// manual Err_Ack 
GVL_Safety.ErrAck := (GVL_Main.key_switch_remote AND GVL_Main.reset_switch);

// manual Restart
GVL_Safety.Restart := (GVL_Main.key_switch_remote AND GVL_Main.start_switch);

ErrAckLog(	Trigger := GVL_Safety.ErrAck,
			OnMessage := 'Safety error was acknowledged.');
			
RestartLog(	Trigger := GVL_Safety.Restart,
			Level := ADSLOG_MSGTYPE_WARN,
			OnMessage := 'Safety was restarted.');

SafetyLog(	Trigger := Error,
			Level := ADSLOG_MSGTYPE_ERROR,
			OnMessage := 'Safety Error! Emergency stop enganged!',
			OffMessage := 'Safety is OK.',
			OffLevel := ADSLOG_MSGTYPE_HINT);
*)

(*
// wait n seconds after Start ...
start_delay(IN := TRUE);
// ... and send ErrAck for n milliseconds
ErrAck_Pulse(IN := (GVL_Safety.State = 2) AND start_delay.Q);

// Error Acknowledgment: Turn key_switch OFF and press STOP 
GVL_Safety.ErrAck := (GVL_Main.key_switch_remote AND GVL_Main.reset_switch)
					OR ErrAck_Pulse.Q
					OR remote_ErrAck;
// detect falling edge 
ErrAck_Trigger(CLK := GVL_Safety.ErrAck);
// send restart pulse on falling edge of ErrAck
restart_pulse(IN := ErrAck_Trigger.Q);

// RESTART Safety after pushing reset or power on delay
GVL_Safety.Restart := (GVL_Main.key_switch_remote AND GVL_Main.start_switch)
 					   OR remote_restart
                       OR restart_pulse.Q;
				
//Error := GVL_Safety.Error OR (GVL_Safety.State <> 1);

//Emergency_stop := NOT GVL_Safety.Stop;

ErrAckLog(	Trigger := GVL_Safety.ErrAck,
			OnMessage := 'Safety error was acknowledged.');
			
RestartLog(	Trigger := GVL_Safety.Restart,
			Level := ADSLOG_MSGTYPE_WARN,
			OnMessage := 'Safety was restarted.');

SafetyLog(	Trigger := Error,
			Level := ADSLOG_MSGTYPE_ERROR,
			OnMessage := 'Safety Error! Emergency stop enganged!',
			OffMessage := 'Safety is OK.',
			OffLevel := ADSLOG_MSGTYPE_HINT);
*)

END_PROGRAM

// ---- POUs/FunctionBlocks/FB_InfoGroup.TcPOU
FUNCTION_BLOCK FB_InfoGroup
VAR_INPUT
	stInfoData	:ST_InfoDataGroup;
END_VAR
VAR_OUTPUT
	sState		:STRING;
END_VAR
VAR
END_VAR

IF stInfoData.usiMapState= 1 THEN
	sState:='RUN';
ELSIF stInfoData.usiMapState= 2 THEN
	sState:='STOP';
ELSIF stInfoData.usiMapState= 3 THEN
	sState:='SAFE';
ELSIF stInfoData.usiMapState= 4 THEN
	sState:='ERROR';
ELSIF stInfoData.usiMapState= 5 THEN
	sState:='RESET';
ELSE
	sState:='Unknown';
END_IF

END_FUNCTION_BLOCK

// ---- POUs/FunctionBlocks/FB_InfoEStop.TcPOU
FUNCTION_BLOCK FB_InfoEStop
VAR_INPUT
	stInfoData		:ST_InfoDataFB;
END_VAR
VAR_OUTPUT
	sState			:STRING;
	sDiag			:STRING;
END_VAR

IF stInfoData.usiMapState= 0 THEN
	sState:='undefined';
ELSIF stInfoData.usiMapState= 1 THEN
	sState:='RUN';
ELSIF stInfoData.usiMapState= 2 THEN
	sState:='STOP';
ELSIF stInfoData.usiMapState= 3 THEN
	sState:='SAFE';
ELSIF stInfoData.usiMapState= 4 THEN
	sState:='ERROR';
ELSIF stInfoData.usiMapState= 5 THEN
	sState:='RESET';
ELSIF stInfoData.usiMapState= 6 THEN
	sState:='START';
ELSIF stInfoData.usiMapState= 8 THEN
	sState:='DELAYOUT';
ELSE
	sState:='Unknown';
END_IF

IF stInfoData.uiMapDiag = 0 THEN
	sDiag:='No error';
ELSIF stInfoData.uiMapDiag.0 THEN
	sDiag:='Discrepancy error input group 1';
ELSIF stInfoData.uiMapDiag.1 THEN
	sDiag:='Discrepancy error input group 2';
ELSIF stInfoData.uiMapDiag.2 THEN
	sDiag:='Discrepancy error input group 3';
ELSIF stInfoData.uiMapDiag.3 THEN
	sDiag:='Discrepancy error input group 4';
ELSIF stInfoData.uiMapDiag.4 THEN
	sDiag:='EDM Error EDM 1';
ELSIF stInfoData.uiMapDiag.5 THEN
	sDiag:='EDM Error EDM 2';
ELSE
	sDiag:='Unknown';
END_IF

END_FUNCTION_BLOCK

// ---- POUs/FunctionBlocks/FB_InfoConnection.TcPOU
FUNCTION_BLOCK FB_InfoConnection
VAR_INPUT
	stInfoData	:ST_InfoDataConnection;
END_VAR
VAR_OUTPUT
	sState		:STRING;
	sDiag		:STRING;
	bChannel1	:BOOL;
	bChannel2	:BOOL;
	bChannel3	:BOOL;
	bChannel4	:BOOL;
END_VAR

IF stInfoData.usiMapState = 100 THEN
	sState:='State Reset';
ELSIF stInfoData.usiMapState = 101 THEN
	sState:='State Session';
ELSIF stInfoData.usiMapState = 102 THEN
	sState:='State Connection';
ELSIF stInfoData.usiMapState = 103 THEN
	sState:='State Parameter';
ELSIF stInfoData.usiMapState = 104 THEN
	sState:='State Data';
ELSIF stInfoData.usiMapState = 105 THEN
	sState:='State Shutdown';
ELSE
	sState:='Error';
END_IF

IF stInfoData.usiMapDiag = 0 THEN
	sDiag:='No error';
ELSIF	stInfoData.usiMapDiag.0 = TRUE THEN
	sDiag:='Invalid Command';
ELSIF	stInfoData.usiMapDiag.1 = TRUE THEN
	sDiag:='Unknown Command';
ELSIF	(stInfoData.usiMapDiag.1 AND stInfoData.usiMapDiag.0)= TRUE THEN
	sDiag:='Invalid Connection ID';
ELSIF	 stInfoData.usiMapDiag.2= TRUE THEN
	sDiag:='Invalid CRC';
ELSIF	(stInfoData.usiMapDiag.0 AND stInfoData.usiMapDiag.2)= TRUE THEN
	sDiag:='Watchdog expired';
ELSIF	(stInfoData.usiMapDiag.1 AND stInfoData.usiMapDiag.2)= TRUE THEN
	sDiag:='Invalid FSoE address';
ELSIF	(stInfoData.usiMapDiag.0 AND stInfoData.usiMapDiag.1 AND stInfoData.usiMapDiag.2)= TRUE THEN
	sDiag:='Invalid data';
ELSIF	stInfoData.usiMapDiag.3= TRUE THEN
	sDiag:='Invalid Com.-Parameter length';
ELSIF	(stInfoData.usiMapDiag.0 AND stInfoData.usiMapDiag.3)= TRUE THEN
	sDiag:='Invalid Com.-Parameter ';
ELSIF	(stInfoData.usiMapDiag.1 AND stInfoData.usiMapDiag.3)= TRUE THEN
	sDiag:='Invalid User.-Parameter length';
ELSIF	(stInfoData.usiMapDiag.0 AND stInfoData.usiMapDiag.1 AND stInfoData.usiMapDiag.3)= TRUE THEN
	sDiag:='Invalid User.-Parameter ';
ELSIF	(stInfoData.usiMapDiag.2 AND stInfoData.usiMapDiag.3)= TRUE THEN
	sDiag:='FSoE Master Reset  ';
ELSIF	stInfoData.usiMapDiag.4= TRUE THEN
	sDiag:='Error by FSoE Slave detected';
ELSIF	stInfoData.usiMapDiag.5= TRUE THEN
	sDiag:='FSoE Slave reports Failsafe value active';
ELSIF	stInfoData.usiMapDiag.6= TRUE THEN
	sDiag:='StartUp';
ELSIF	stInfoData.usiMapDiag.7= TRUE THEN
	sDiag:='FSoE Master reports Failsafe value active';
ELSE
	sDiag:='Error';
END_IF

(*Signals*)
bChannel1 := stInfoData.bySignal.0;
bChannel2 := stInfoData.bySignal.1;
bChannel3 := stInfoData.bySignal.2;
bChannel4 := stInfoData.bySignal.3;

END_FUNCTION_BLOCK

// ---- GlobalTextList.TcGTLO
TEXTLIST GlobalTextList
  785 = 'Azimuth:'
  798 = 'Brake closed'
  396 = 'Brake open'
  272 = 'busy'
  41 = 'Close brake'
  815 = 'Derotator:'
  524 = 'Diag: %s'
  101 = 'EL1904'
  761 = 'EL2904'
  409 = 'Elevation:'
  894 = 'Enable'
  868 = 'ErrAck'
  879 = 'Error'
  225 = 'Estop: %s'
  548 = 'GoHome'
  867 = 'GoTo'
  33 = 'Oil cold'
  995 = 'Oil high'
  856 = 'Oil hot'
  768 = 'Oil low'
  481 = 'Oil pressure OK'
  498 = 'Oil warning'
  482 = 'Open brake'
  352 = 'Override Start Pump'
  744 = 'Override Start Sucction'
  606 = 'Override stop pump'
  273 = 'park'
  919 = 'Power'
  523 = 'Pump running'
  120 = 'ready'
  685 = 'Reset'
  789 = 'Restart'
  104 = 'Safety Diag%s'
  521 = 'Safety Diag: %s'
  672 = 'Safety State: %s'
  777 = 'slew'
  717 = 'sliding'
  809 = 'State: %s'
  328 = 'STO ErrAck:'
  540 = 'STO Reset:'
  488 = 'STO:'
  572 = 'Stop'
  155 = 'stopped'
  782 = 'Sucction running'
  704 = 'Succtionrunning'
  362 = 'track'
  364 = 'tracking'
END_TEXTLIST

// ---- VISUs/Safety.TcVIS
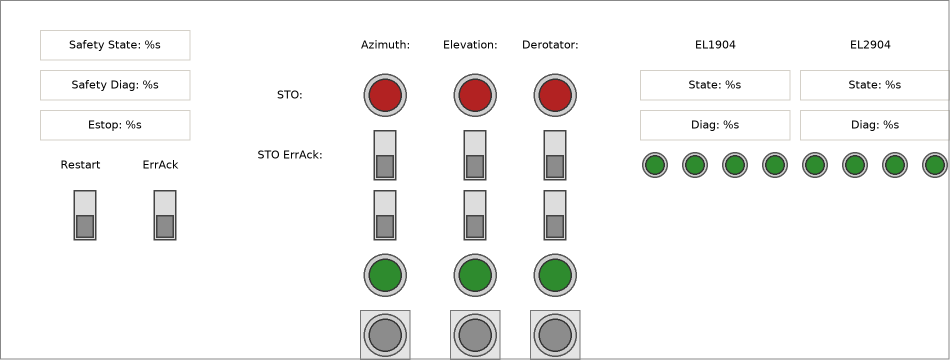
VISUALIZATION Safety  // 950x360
    Label (340,30 91x30), "Azimuth:"
    Lamp1 (360,70 50x50), variable: GVL_Telescope.Azimuth_sto, style: Lamp-Lamp1-Red
    Label (430,30 81x30), "Elevation:"
    Lamp1 (450,70 50x50), variable: GVL_Telescope.Elevation_sto, style: Lamp-Lamp1-Red
    Label (510,30 81x30), "Derotator:"
    Lamp1 (530,70 50x50), variable: GVL_Telescope.Derotator_sto, style: Lamp-Lamp1-Red
    Label (240,80 100x30), "STO:"
    Lamp1 (360,250 50x50), variable: AzimuthElevationControl.ready, style: Lamp-Lamp1-Green
    Lamp1 (450,250 50x50), variable: ElevationControl.Ready, style: Lamp-Lamp1-Green
    Lamp1 (530,250 50x50), style: Lamp-Lamp1-Green
    PushSwitch (360,310 50x50), variable: AzimuthElevationControl.Reset, behaviour: TAP, style: Switch-PushSwitch-Gray
    PushSwitch (450,310 50x50), variable: ElevationControl.reset, behaviour: TAP, style: Switch-PushSwitch-Gray
    PushSwitch (530,310 50x50), behaviour: TAP, style: Switch-PushSwitch-Gray
    DipSwitch (360,190 50x50), variable: AzimuthElevationControl.Enable, behaviour: TOGGLE, style: Switch-DipSwitch-Gray
    DipSwitch (450,190 50x50), variable: ElevationControl.enable, behaviour: TOGGLE, style: Switch-DipSwitch-Gray
    DipSwitch (530,190 50x50), variable: DerotatorControl.enable, behaviour: TOGGLE, style: Switch-DipSwitch-Gray
    DipSwitch (60,190 50x50), variable: GVL_Safety.Restart, behaviour: TOGGLE, style: Switch-DipSwitch-Gray
    DipSwitch (530,130 50x50), variable: GVL_Safety.Reset_STO_Derotator, behaviour: TOGGLE, style: Switch-DipSwitch-Gray
    DipSwitch (360,130 50x50), variable: GVL_Safety.Reset_STO_Azimuth, behaviour: TOGGLE, style: Switch-DipSwitch-Gray
    DipSwitch (450,130 50x50), variable: GVL_Safety.Reset_STO_Elevation, behaviour: TOGGLE, style: Switch-DipSwitch-Gray
    Label (240,140 100x30), "STO ErrAck:"
    Label (40,150 81x30), "Restart"
    DipSwitch (140,190 50x50), variable: GVL_Safety.ErrAck, behaviour: TOGGLE, style: Switch-DipSwitch-Gray
    Label (120,150 81x30), "ErrAck"
    Textfield (40,30 150x30), "Safety State: %s", text variable: SafetyHandling.fbInfoEStop1.sState, input disabled if: TRUE
    Textfield (40,110 150x30), "Estop: %s", text variable: SafetyHandling.fbInfoEStop1.sState, input disabled if: TRUE
    Textfield (40,70 150x30), "Safety Diag: %s", text variable: SafetyHandling.fbInfoEStop1.sDiag, input disabled if: TRUE
    Label (670,30 91x30), "EL1904"
    Label (830,30 81x30), "EL2904"
    Textfield (640,70 150x30), "State: %s", text variable: SafetyHandling.fbInfoSafetyIn.sState, input disabled if: TRUE
    Textfield (640,110 150x30), "Diag: %s", text variable: SafetyHandling.fbInfoSafetyIn.sDiag, input disabled if: TRUE
    Textfield (800,70 150x30), "State: %s", text variable: SafetyHandling.fbInfoSafetyOut.sState, input disabled if: TRUE
    Textfield (800,110 150x30), "Diag: %s", text variable: SafetyHandling.fbInfoSafetyOut.sDiag, input disabled if: TRUE
    Lamp1 (640,150 30x30), variable: SafetyHandling.bSafetyInCh1, style: Lamp-Lamp1-Green
    Lamp1 (680,150 30x30), variable: SafetyHandling.bSafetyInCh2, style: Lamp-Lamp1-Green
    Lamp1 (720,150 30x30), variable: SafetyHandling.bSafetyInCh3, style: Lamp-Lamp1-Green
    Lamp1 (760,150 30x30), variable: SafetyHandling.bSafetyInCh4, style: Lamp-Lamp1-Green
    Lamp1 (800,150 30x30), variable: SafetyHandling.bSafetyInCh1, style: Lamp-Lamp1-Green
    Lamp1 (840,150 30x30), variable: SafetyHandling.bSafetyInCh2, style: Lamp-Lamp1-Green
    Lamp1 (880,150 30x30), variable: SafetyHandling.bSafetyInCh3, style: Lamp-Lamp1-Green
    Lamp1 (920,150 30x30), variable: SafetyHandling.bSafetyInCh4, style: Lamp-Lamp1-Green
END_VISUALIZATION

// ---- VISUs/Visualization.TcVIS
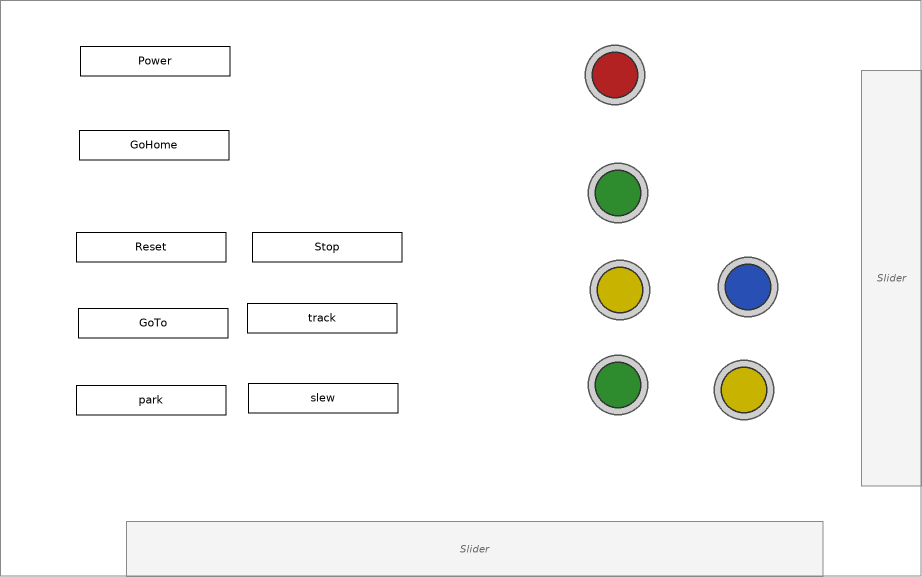
VISUALIZATION Visualization  // 922x577
    RoundedRectangle (80,46 150x30), "Power", colour toggle: TelescopeControl.power
        toggle TelescopeControl.power
    Rectangle (79,130 150x30), "GoHome", colour toggle: TelescopeControl.gohome
        toggle TelescopeControl.gohome
    Lamp1 (580,40 70x70), tooltip "Error", variable: TelescopeControl.error, style: Lamp-Lamp1-Red
    Lamp1 (583,158 70x70), tooltip "ready", variable: TelescopeControl.ready, style: Lamp-Lamp1-Green
    Rectangle (76,232 150x30), "Reset", colour toggle: TelescopeControl.reset
        toggle TelescopeControl.reset
    RoundedRectangle (78,308 150x30), "GoTo", colour toggle: TelescopeControl.goto
        toggle TelescopeControl.goto
    Lamp1 (585,255 70x70), tooltip "sliding", variable: TelescopeControl.sliding, style: Lamp-Lamp1-Yellow
    RoundedRectangle (76,385 150x30), "park", colour toggle: TelescopeControl.park
        toggle TelescopeControl.park
    Lamp1 (583,350 70x70), tooltip "stopped", variable: TelescopeControl.Safetypped, style: Lamp-Lamp1-Green
    Slider (126,521 697x56), variable: TelescopeControl.rightascension, scale 0..360
    Slider (861,70 61x416), variable: TelescopeControl.declination, scale -90..90
    Lamp1 (713,252 70x70), tooltip "tracking", variable: TelescopeControl.tracking, style: Lamp-Lamp1-Blue
    RoundedRectangle (247,303 150x30), "track", colour toggle: TelescopeControl.track
        toggle TelescopeControl.track
    RoundedRectangle (248,383 150x30), "slew", colour toggle: TelescopeControl.slew
        toggle TelescopeControl.slew
    Lamp1 (709,355 70x70), tooltip "busy", variable: TelescopeControl.busy, style: Lamp-Lamp1-Yellow
    RoundedRectangle (252,232 150x30), "Stop", colour toggle: TelescopeControl.Safetyp
        toggle TelescopeControl.stop
END_VISUALIZATION
